# EPICS StreamDevice protocol: merlot/merlot.proto
Terminator = LF;

GetVersion {
	out "v";
	in "v %#s";
}

Enable1 {
	out "e0 %d";
	@init {
		out "e";
		in "e %d %*d %*d %*d %*d %*d %*d %*d";
	}
}
Enable2 {
	out "e1 %d";
	@init {
		out "e";
		in "e %*d %d %*d %*d %*d %*d %*d %*d";
	}
}
Enable3 {
	out "e2 %d";
	@init {
		out "e";
		in "e %*d %*d %d %*d %*d %*d %*d %*d";
	}
}
Enable4 {
	out "e3 %d";
	@init {
		out "e";
		in "e %*d %*d %*d %d %*d %*d %*d %*d";
	}
}
Enable5 {
	out "e4 %d";
	@init {
		out "e";
		in "e %*d %*d %*d %*d %d %*d %*d %*d";
	}
}
Enable6 {
	out "e5 %d";
	@init {
		out "e";
		in "e %*d %*d %*d %*d %*d %d %*d %*d";
	}
}
Enable7 {
	out "e6 %d";
	@init {
		out "e";
		in "e %*d %*d %*d %*d %*d %*d %d %*d";
	}
}
Enable8 {
	out "e7 %d";
	@init {
		out "e";
		in "e %*d %*d %*d %*d %*d %*d %*d %d";
	}
}

GetCurrentTemp1 {
	out "r";
	in "r %f %*f %*d %*d %*d %*f %*f %*d %*d %*d %*f %*f %*d %*d %*d %*f %*f %*d %*d %*d %*f %*f %*d %*d %*d %*f %*f %*d %*d %*d %*f %*f %*d %*d %*d %*f %*f %*d %*d %*d";
}
GetDutyCycle1   { in "r %*f %f %*d %*d %*d %*f %*f %*d %*d %*d %*f %*f %*d %*d %*d %*f %*f %*d %*d %*d %*f %*f %*d %*d %*d %*f %*f %*d %*d %*d %*f %*f %*d %*d %*d %*f %*f %*d %*d %*d"; }
GetPTerm1       { in "r %*f %*f %d %*d %*d %*f %*f %*d %*d %*d %*f %*f %*d %*d %*d %*f %*f %*d %*d %*d %*f %*f %*d %*d %*d %*f %*f %*d %*d %*d %*f %*f %*d %*d %*d %*f %*f %*d %*d %*d"; }
GetITerm1       { in "r %*f %*f %*d %d %*d %*f %*f %*d %*d %*d %*f %*f %*d %*d %*d %*f %*f %*d %*d %*d %*f %*f %*d %*d %*d %*f %*f %*d %*d %*d %*f %*f %*d %*d %*d %*f %*f %*d %*d %*d"; }
GetDTerm1       { in "r %*f %*f %*d %*d %d %*f %*f %*d %*d %*d %*f %*f %*d %*d %*d %*f %*f %*d %*d %*d %*f %*f %*d %*d %*d %*f %*f %*d %*d %*d %*f %*f %*d %*d %*d %*f %*f %*d %*d %*d"; }
GetCurrentTemp2 { in "r %*f %*f %*d %*d %*d %f %*f %*d %*d %*d %*f %*f %*d %*d %*d %*f %*f %*d %*d %*d %*f %*f %*d %*d %*d %*f %*f %*d %*d %*d %*f %*f %*d %*d %*d %*f %*f %*d %*d %*d"; }
GetDutyCycle2   { in "r %*f %*f %*d %*d %*d %*f %f %*d %*d %*d %*f %*f %*d %*d %*d %*f %*f %*d %*d %*d %*f %*f %*d %*d %*d %*f %*f %*d %*d %*d %*f %*f %*d %*d %*d %*f %*f %*d %*d %*d"; }
GetPTerm2       { in "r %*f %*f %*d %*d %*d %*f %*f %d %*d %*d %*f %*f %*d %*d %*d %*f %*f %*d %*d %*d %*f %*f %*d %*d %*d %*f %*f %*d %*d %*d %*f %*f %*d %*d %*d %*f %*f %*d %*d %*d"; }
GetITerm2       { in "r %*f %*f %*d %*d %*d %*f %*f %*d %d %*d %*f %*f %*d %*d %*d %*f %*f %*d %*d %*d %*f %*f %*d %*d %*d %*f %*f %*d %*d %*d %*f %*f %*d %*d %*d %*f %*f %*d %*d %*d"; }
GetDTerm2       { in "r %*f %*f %*d %*d %*d %*f %*f %*d %*d %d %*f %*f %*d %*d %*d %*f %*f %*d %*d %*d %*f %*f %*d %*d %*d %*f %*f %*d %*d %*d %*f %*f %*d %*d %*d %*f %*f %*d %*d %*d"; }
GetCurrentTemp3 { in "r %*f %*f %*d %*d %*d %*f %*f %*d %*d %*d %f %*f %*d %*d %*d %*f %*f %*d %*d %*d %*f %*f %*d %*d %*d %*f %*f %*d %*d %*d %*f %*f %*d %*d %*d %*f %*f %*d %*d %*d"; }
GetDutyCycle3   { in "r %*f %*f %*d %*d %*d %*f %*f %*d %*d %*d %*f %f %*d %*d %*d %*f %*f %*d %*d %*d %*f %*f %*d %*d %*d %*f %*f %*d %*d %*d %*f %*f %*d %*d %*d %*f %*f %*d %*d %*d"; }
GetPTerm3       { in "r %*f %*f %*d %*d %*d %*f %*f %*d %*d %*d %*f %*f %d %*d %*d %*f %*f %*d %*d %*d %*f %*f %*d %*d %*d %*f %*f %*d %*d %*d %*f %*f %*d %*d %*d %*f %*f %*d %*d %*d"; }
GetITerm3       { in "r %*f %*f %*d %*d %*d %*f %*f %*d %*d %*d %*f %*f %*d %d %*d %*f %*f %*d %*d %*d %*f %*f %*d %*d %*d %*f %*f %*d %*d %*d %*f %*f %*d %*d %*d %*f %*f %*d %*d %*d"; }
GetDTerm3       { in "r %*f %*f %*d %*d %*d %*f %*f %*d %*d %*d %*f %*f %*d %*d %d %*f %*f %*d %*d %*d %*f %*f %*d %*d %*d %*f %*f %*d %*d %*d %*f %*f %*d %*d %*d %*f %*f %*d %*d %*d"; }
GetCurrentTemp4 { in "r %*f %*f %*d %*d %*d %*f %*f %*d %*d %*d %*f %*f %*d %*d %*d %f %*f %*d %*d %*d %*f %*f %*d %*d %*d %*f %*f %*d %*d %*d %*f %*f %*d %*d %*d %*f %*f %*d %*d %*d"; }
GetDutyCycle4   { in "r %*f %*f %*d %*d %*d %*f %*f %*d %*d %*d %*f %*f %*d %*d %*d %*f %f %*d %*d %*d %*f %*f %*d %*d %*d %*f %*f %*d %*d %*d %*f %*f %*d %*d %*d %*f %*f %*d %*d %*d"; }
GetPTerm4       { in "r %*f %*f %*d %*d %*d %*f %*f %*d %*d %*d %*f %*f %*d %*d %*d %*f %*f %d %*d %*d %*f %*f %*d %*d %*d %*f %*f %*d %*d %*d %*f %*f %*d %*d %*d %*f %*f %*d %*d %*d"; }
GetITerm4       { in "r %*f %*f %*d %*d %*d %*f %*f %*d %*d %*d %*f %*f %*d %*d %*d %*f %*f %*d %d %*d %*f %*f %*d %*d %*d %*f %*f %*d %*d %*d %*f %*f %*d %*d %*d %*f %*f %*d %*d %*d"; }
GetDTerm4       { in "r %*f %*f %*d %*d %*d %*f %*f %*d %*d %*d %*f %*f %*d %*d %*d %*f %*f %*d %*d %d %*f %*f %*d %*d %*d %*f %*f %*d %*d %*d %*f %*f %*d %*d %*d %*f %*f %*d %*d %*d"; }
GetCurrentTemp5 { in "r %*f %*f %*d %*d %*d %*f %*f %*d %*d %*d %*f %*f %*d %*d %*d %*f %*f %*d %*d %*d %f %*f %*d %*d %*d %*f %*f %*d %*d %*d %*f %*f %*d %*d %*d %*f %*f %*d %*d %*d"; }
GetDutyCycle5   { in "r %*f %*f %*d %*d %*d %*f %*f %*d %*d %*d %*f %*f %*d %*d %*d %*f %*f %*d %*d %*d %*f %f %*d %*d %*d %*f %*f %*d %*d %*d %*f %*f %*d %*d %*d %*f %*f %*d %*d %*d"; }
GetPTerm5       { in "r %*f %*f %*d %*d %*d %*f %*f %*d %*d %*d %*f %*f %*d %*d %*d %*f %*f %*d %*d %*d %*f %*f %d %*d %*d %*f %*f %*d %*d %*d %*f %*f %*d %*d %*d %*f %*f %*d %*d %*d"; }
GetITerm5       { in "r %*f %*f %*d %*d %*d %*f %*f %*d %*d %*d %*f %*f %*d %*d %*d %*f %*f %*d %*d %*d %*f %*f %*d %d %*d %*f %*f %*d %*d %*d %*f %*f %*d %*d %*d %*f %*f %*d %*d %*d"; }
GetDTerm5       { in "r %*f %*f %*d %*d %*d %*f %*f %*d %*d %*d %*f %*f %*d %*d %*d %*f %*f %*d %*d %*d %*f %*f %*d %*d %d %*f %*f %*d %*d %*d %*f %*f %*d %*d %*d %*f %*f %*d %*d %*d"; }
GetCurrentTemp6 { in "r %*f %*f %*d %*d %*d %*f %*f %*d %*d %*d %*f %*f %*d %*d %*d %*f %*f %*d %*d %*d %*f %*f %*d %*d %*d %f %*f %*d %*d %*d %*f %*f %*d %*d %*d %*f %*f %*d %*d %*d"; }
GetDutyCycle6   { in "r %*f %*f %*d %*d %*d %*f %*f %*d %*d %*d %*f %*f %*d %*d %*d %*f %*f %*d %*d %*d %*f %*f %*d %*d %*d %*f %f %*d %*d %*d %*f %*f %*d %*d %*d %*f %*f %*d %*d %*d"; }
GetPTerm6       { in "r %*f %*f %*d %*d %*d %*f %*f %*d %*d %*d %*f %*f %*d %*d %*d %*f %*f %*d %*d %*d %*f %*f %*d %*d %*d %*f %*f %d %*d %*d %*f %*f %*d %*d %*d %*f %*f %*d %*d %*d"; }
GetITerm6       { in "r %*f %*f %*d %*d %*d %*f %*f %*d %*d %*d %*f %*f %*d %*d %*d %*f %*f %*d %*d %*d %*f %*f %*d %*d %*d %*f %*f %*d %d %*d %*f %*f %*d %*d %*d %*f %*f %*d %*d %*d"; }
GetDTerm6       { in "r %*f %*f %*d %*d %*d %*f %*f %*d %*d %*d %*f %*f %*d %*d %*d %*f %*f %*d %*d %*d %*f %*f %*d %*d %*d %*f %*f %*d %*d %d %*f %*f %*d %*d %*d %*f %*f %*d %*d %*d"; }
GetCurrentTemp7 { in "r %*f %*f %*d %*d %*d %*f %*f %*d %*d %*d %*f %*f %*d %*d %*d %*f %*f %*d %*d %*d %*f %*f %*d %*d %*d %*f %*f %*d %*d %*d %f %*f %*d %*d %*d %*f %*f %*d %*d %*d"; }
GetDutyCycle7   { in "r %*f %*f %*d %*d %*d %*f %*f %*d %*d %*d %*f %*f %*d %*d %*d %*f %*f %*d %*d %*d %*f %*f %*d %*d %*d %*f %*f %*d %*d %*d %*f %f %*d %*d %*d %*f %*f %*d %*d %*d"; }
GetPTerm7       { in "r %*f %*f %*d %*d %*d %*f %*f %*d %*d %*d %*f %*f %*d %*d %*d %*f %*f %*d %*d %*d %*f %*f %*d %*d %*d %*f %*f %*d %*d %*d %*f %*f %d %*d %*d %*f %*f %*d %*d %*d"; }
GetITerm7       { in "r %*f %*f %*d %*d %*d %*f %*f %*d %*d %*d %*f %*f %*d %*d %*d %*f %*f %*d %*d %*d %*f %*f %*d %*d %*d %*f %*f %*d %*d %*d %*f %*f %*d %d %*d %*f %*f %*d %*d %*d"; }
GetDTerm7       { in "r %*f %*f %*d %*d %*d %*f %*f %*d %*d %*d %*f %*f %*d %*d %*d %*f %*f %*d %*d %*d %*f %*f %*d %*d %*d %*f %*f %*d %*d %*d %*f %*f %*d %*d %d %*f %*f %*d %*d %*d"; }
GetCurrentTemp8 { in "r %*f %*f %*d %*d %*d %*f %*f %*d %*d %*d %*f %*f %*d %*d %*d %*f %*f %*d %*d %*d %*f %*f %*d %*d %*d %*f %*f %*d %*d %*d %*f %*f %*d %*d %*d %f %*f %*d %*d %*d"; }
GetDutyCycle8   { in "r %*f %*f %*d %*d %*d %*f %*f %*d %*d %*d %*f %*f %*d %*d %*d %*f %*f %*d %*d %*d %*f %*f %*d %*d %*d %*f %*f %*d %*d %*d %*f %*f %*d %*d %*d %*f %f %*d %*d %*d"; }
GetPTerm8       { in "r %*f %*f %*d %*d %*d %*f %*f %*d %*d %*d %*f %*f %*d %*d %*d %*f %*f %*d %*d %*d %*f %*f %*d %*d %*d %*f %*f %*d %*d %*d %*f %*f %*d %*d %*d %*f %*f %d %*d %*d"; }
GetITerm8       { in "r %*f %*f %*d %*d %*d %*f %*f %*d %*d %*d %*f %*f %*d %*d %*d %*f %*f %*d %*d %*d %*f %*f %*d %*d %*d %*f %*f %*d %*d %*d %*f %*f %*d %*d %*d %*f %*f %*d %d %*d"; }
GetDTerm8       { in "r %*f %*f %*d %*d %*d %*f %*f %*d %*d %*d %*f %*f %*d %*d %*d %*f %*f %*d %*d %*d %*f %*f %*d %*d %*d %*f %*f %*d %*d %*d %*f %*f %*d %*d %*d %*f %*f %*d %*d %d"; }

SetMaxDutyCycle1 {
	out "m0 %d";
	@init {
		out "m";
		in "m %d %*d %*d %*d %*d %*d %*d %*d";
	}
}
SetMaxDutyCycle2 {
	out "m1 %d";
	@init {
		out "m";
		in "m %*d %d %*d %*d %*d %*d %*d %*d";
	}
}
SetMaxDutyCycle3 {
	out "m2 %d";
	@init {
		out "m";
		in "m %*d %*d %d %*d %*d %*d %*d %*d";
	}
}
SetMaxDutyCycle4 {
	out "m3 %d";
	@init {
		out "m";
		in "m %*d %*d %*d %d %*d %*d %*d %*d";
	}
}
SetMaxDutyCycle5 {
	out "m4 %d";
	@init {
		out "m";
		in "m %*d %*d %*d %*d %d %*d %*d %*d";
	}
}
SetMaxDutyCycle6 {
	out "m5 %d";
	@init {
		out "m";
		in "m %*d %*d %*d %*d %*d %d %*d %*d";
	}
}
SetMaxDutyCycle7 {
	out "m6 %d";
	@init {
		out "m";
		in "m %*d %*d %*d %*d %*d %*d %d %*d";
	}
}
SetMaxDutyCycle8 {
	out "m7 %d";
	@init {
		out "m";
		in "m %*d %*d %*d %*d %*d %*d %*d %d";
	}
}
SetDesiredTemp1 {
	out "d0 %f";
	@init {
		out "d";
		in "d %f %*f %*f %*f %*f %*f %*f %*f";
	}
}
SetDesiredTemp2 {
	out "d1 %f";
	@init {
		out "d";
		in "d %*f %f %*f %*f %*f %*f %*f %*f";
	}
}
SetDesiredTemp3 {
	out "d2 %f";
	@init {
		out "d";
		in "d %*f %*f %f %*f %*f %*f %*f %*f";
	}
}
SetDesiredTemp4 {
	out "d3 %f";
	@init {
		out "d";
		in "d %*f %*f %*f %f %*f %*f %*f %*f";
	}
}
SetDesiredTemp5 {
	out "d4 %f";
	@init {
		out "d";
		in "d %*f %*f %*f %*f %f %*f %*f %*f";
	}
}
SetDesiredTemp6 {
	out "d5 %f";
	@init {
		out "d";
		in "d %*f %*f %*f %*f %*f %f %*f %*f";
	}
}
SetDesiredTemp7 {
	out "d6 %f";
	@init {
		out "d";
		in "d %*f %*f %*f %*f %*f %*f %f %*f";
	}
}
SetDesiredTemp8 {
	out "d7 %f";
	@init {
		out "d";
		in "d %*f %*f %*f %*f %*f %*f %*f %f";
	}
}

SetP1 { out ""; @init { out "p"; in "p %x %*x %*x %*x %*x %*x %*x %*x %*x %*x %*x %*x %*x %*x %*x %*x %*x %*x %*x %*x %*x %*x %*x %*x"; } }
SetI1 { out ""; @init { out "p"; in "p %*x %x %*x %*x %*x %*x %*x %*x %*x %*x %*x %*x %*x %*x %*x %*x %*x %*x %*x %*x %*x %*x %*x %*x"; } }
SetD1 { out ""; @init { out "p"; in "p %*x %*x %x %*x %*x %*x %*x %*x %*x %*x %*x %*x %*x %*x %*x %*x %*x %*x %*x %*x %*x %*x %*x %*x"; } }
SetPID1 {
	out "p0 %(A)x %(B)x %(C)x";
}

SetP2 { out ""; @init { out "p"; in "p %*x %*x %*x %x %*x %*x %*x %*x %*x %*x %*x %*x %*x %*x %*x %*x %*x %*x %*x %*x %*x %*x %*x %*x"; } }
SetI2 { out ""; @init { out "p"; in "p %*x %*x %*x %*x %x %*x %*x %*x %*x %*x %*x %*x %*x %*x %*x %*x %*x %*x %*x %*x %*x %*x %*x %*x"; } }
SetD2 { out ""; @init { out "p"; in "p %*x %*x %*x %*x %*x %x %*x %*x %*x %*x %*x %*x %*x %*x %*x %*x %*x %*x %*x %*x %*x %*x %*x %*x"; } }
SetPID2 {
	out "p1 %(A)x %(B)x %(C)x";
}

SetP3 { out ""; @init { out "p"; in "p %*x %*x %*x %*x %*x %*x %x %*x %*x %*x %*x %*x %*x %*x %*x %*x %*x %*x %*x %*x %*x %*x %*x %*x"; } }
SetI3 { out ""; @init { out "p"; in "p %*x %*x %*x %*x %*x %*x %*x %x %*x %*x %*x %*x %*x %*x %*x %*x %*x %*x %*x %*x %*x %*x %*x %*x"; } }
SetD3 { out ""; @init { out "p"; in "p %*x %*x %*x %*x %*x %*x %*x %*x %x %*x %*x %*x %*x %*x %*x %*x %*x %*x %*x %*x %*x %*x %*x %*x"; } }
SetPID3 {
	out "p2 %(A)x %(B)x %(C)x";
}

SetP4 { out ""; @init { out "p"; in "p %*x %*x %*x %*x %*x %*x %*x %*x %*x %x %*x %*x %*x %*x %*x %*x %*x %*x %*x %*x %*x %*x %*x %*x"; } }
SetI4 { out ""; @init { out "p"; in "p %*x %*x %*x %*x %*x %*x %*x %*x %*x %*x %x %*x %*x %*x %*x %*x %*x %*x %*x %*x %*x %*x %*x %*x"; } }
SetD4 { out ""; @init { out "p"; in "p %*x %*x %*x %*x %*x %*x %*x %*x %*x %*x %*x %x %*x %*x %*x %*x %*x %*x %*x %*x %*x %*x %*x %*x"; } }
SetPID4 {
	out "p3 %(A)x %(B)x %(C)x";
}

SetP5 { out ""; @init { out "p"; in "p %*x %*x %*x %*x %*x %*x %*x %*x %*x %*x %*x %*x %x %*x %*x %*x %*x %*x %*x %*x %*x %*x %*x %*x"; } }
SetI5 { out ""; @init { out "p"; in "p %*x %*x %*x %*x %*x %*x %*x %*x %*x %*x %*x %*x %*x %x %*x %*x %*x %*x %*x %*x %*x %*x %*x %*x"; } }
SetD5 { out ""; @init { out "p"; in "p %*x %*x %*x %*x %*x %*x %*x %*x %*x %*x %*x %*x %*x %*x %x %*x %*x %*x %*x %*x %*x %*x %*x %*x"; } }
SetPID5 {
	out "p4 %(A)x %(B)x %(C)x";
}

SetP6 { out ""; @init { out "p"; in "p %*x %*x %*x %*x %*x %*x %*x %*x %*x %*x %*x %*x %*x %*x %*x %x %*x %*x %*x %*x %*x %*x %*x %*x"; } }
SetI6 { out ""; @init { out "p"; in "p %*x %*x %*x %*x %*x %*x %*x %*x %*x %*x %*x %*x %*x %*x %*x %*x %x %*x %*x %*x %*x %*x %*x %*x"; } }
SetD6 { out ""; @init { out "p"; in "p %*x %*x %*x %*x %*x %*x %*x %*x %*x %*x %*x %*x %*x %*x %*x %*x %*x %x %*x %*x %*x %*x %*x %*x"; } }
SetPID6 {
	out "p5 %(A)x %(B)x %(C)x";
}

SetP7 { out ""; @init { out "p"; in "p %*x %*x %*x %*x %*x %*x %*x %*x %*x %*x %*x %*x %*x %*x %*x %*x %*x %*x %x %*x %*x %*x %*x %*x"; } }
SetI7 { out ""; @init { out "p"; in "p %*x %*x %*x %*x %*x %*x %*x %*x %*x %*x %*x %*x %*x %*x %*x %*x %*x %*x %*x %x %*x %*x %*x %*x"; } }
SetD7 { out ""; @init { out "p"; in "p %*x %*x %*x %*x %*x %*x %*x %*x %*x %*x %*x %*x %*x %*x %*x %*x %*x %*x %*x %*x %x %*x %*x %*x"; } }
SetPID7 {
	out "p6 %(A)x %(B)x %(C)x";
}

SetP8 { out ""; @init { out "p"; in "p %*x %*x %*x %*x %*x %*x %*x %*x %*x %*x %*x %*x %*x %*x %*x %*x %*x %*x %*x %*x %*x %x %*x %*x"; } }
SetI8 { out ""; @init { out "p"; in "p %*x %*x %*x %*x %*x %*x %*x %*x %*x %*x %*x %*x %*x %*x %*x %*x %*x %*x %*x %*x %*x %*x %x %*x"; } }
SetD8 { out ""; @init { out "p"; in "p %*x %*x %*x %*x %*x %*x %*x %*x %*x %*x %*x %*x %*x %*x %*x %*x %*x %*x %*x %*x %*x %*x %*x %x"; } }
SetPID8 {
	out "p7 %(A)x %(B)x %(C)x";
}
